FUNCTION alg_M_mode_a_Dstartled : BOOL
VAR_INPUT
	state: STATE;
END_VAR

alg_M_mode_a_Dstartled := (state.dvar_M_mode) = (elit_on);

END_FUNCTION

(* stored: Version 1.1.0.1, ProductVersion 3.1.4022.18
   POU alg_M_mode_a_Dstartled: Id {e97a5acd-d5d2-4ed0-8d98-beb3d47e7a72}, SpecialFunc None *)
